GLOBALCONSTANTS AID_WSSC (* Working set special controls object attribute ids *)
  (* Standard: 61499-1; Description: Copyright (c) 2023 HR Agrartechnik GmbH This program and the accompanying materials are made available under the terms of the Eclipse Public License 2.0 which is available at https://www.eclipse.org/legal/epl-2.0/ SPDX-License-Identifier: EPL-2.0 *)
  (* Version 1.0, 2026-06-20, Franz Höpfinger, HR Agrartechnik GmbH *)
  PACKAGE isobus::UT::Q::const::AID;
  IMPORT eclipse4diac::core::TypeHash;
  VAR_GLOBAL CONSTANT
    NUMOFBYTES : USINT := USINT#1; (* 1: AID_WSSC_NUMOFBYTES - Number of bytes to follow in this object. *)
    COLOUR_MAP : USINT := USINT#2; (* 2: AID_WSSC_COLOUR_MAP - Object ID of a Colour Map object, or NULL. *)
    COLOUR_PALETTE : USINT := USINT#3; (* 3: AID_WSSC_COLOUR_PALETTE - Object ID of a Colour Palette object, or NULL. *)
  END_VAR
END_GLOBALCONSTANTS
